(* CODESYS project PLC_Project_RECOVERED_2025-07-25T08-23-59.project

Project tree, tasks and I/O mapping:
  Device : CODESYS Control Win V3 x64, CODESYS, version 3.5.21.10
    application Application
      libraries: Standard, 3.5.18.0 (System)
      task MainTask (cyclic, interval t#20ms, priority 1) calls PLC_PRG
      section4_Method/
        function block sec4_Motor [ST]: OvldSet, StopManual, Stop, OvldReset, StartManual, Start
        program sec4_Main [ST]
      program PLC_PRG [ST]
      section2_BasicST/
        Lecture1_StandardFunction/
          program Lecture1_StandardFunction [ST]
        Exercise1/
          program Exercise1 [ST]
        Lecture2_Finite State Machine/
          program Lecture2_FiniteStateMachine [ST]
        Lecture3_Array/
          program Lecture3_Array [ST]
          function CheckFault [ST]
      section3_Class/
        Lecture1_Class/
          program POU_Class_Lecture1 [ST]
          function block Motor [ST]
          data type DUT_MotorInputVar
          data type DUT_MotorOutputVar
        Exercise1/
          data type MotorO
          data type MotorI
          program POU_Class_Exercise1 [ST]
          function block MotorEquip [ST]
*)

// Device/Application/section3_Class/Exercise1/MotorO
TYPE MotorO :
STRUCT
	Coil : BOOL;
END_STRUCT
END_TYPE

// Device/Application/section3_Class/Exercise1/MotorI
TYPE MotorI :
STRUCT
	Start : BOOL;
	Stop  : BOOL;
	OverLoad : BOOL;
	WaitTime :TIME;
 
END_STRUCT
END_TYPE

// Device/Application/section3_Class/Lecture1_Class/DUT_MotorInputVar
TYPE DUT_MotorInputVar :
	
STRUCT
	Start : BOOL;
	Stop : BOOL;
	Overload : BOOL;
END_STRUCT


END_TYPE

// Device/Application/section3_Class/Lecture1_Class/DUT_MotorOutputVar
TYPE DUT_MotorOutputVar :
	
STRUCT
	Coil : BOOL;
END_STRUCT

END_TYPE

// Device/Application/PLC_PRG
PROGRAM PLC_PRG
VAR
	Motor1 : Motor;
END_VAR

//Lecture1_StandardFunction();
//Lecture2_FiniteStateMachine();
//Lecture3_Array();
//Exercise1();
//POU_Class_Lecture1();
//POU_Class_Exercise1();
sec4_Main();

END_PROGRAM

// Device/Application/section2_BasicST/Lecture1_StandardFunction/Lecture1_StandardFunction
PROGRAM Lecture1_StandardFunction
VAR
	Start : BOOL;
	Stop : BOOL;
	Motor1 : BOOL;
	Motor2 : BOOL;
	
	Timer1 : TON;
	ElapsedTime: TIME;
	
	Reset : BOOL;
	StartTrigger : R_TRIG;
	StopTrigger : R_TRIG;
END_VAR


StartTrigger(CLK:= Start);
StopTrigger(CLK:= Stop);


IF StartTrigger.Q THEN
	Motor1 := TRUE;
END_IF


IF Motor1 THEN	
	Timer1(IN:=TRUE ,PT:=T#10S ,
	   ET=>ElapsedTime );	   
END_IF

IF Timer1.Q THEN
	Motor2 := TRUE;
END_IF
	  


IF StopTrigger.Q THEN
	Timer1(IN:=FALSE ,PT:=T#5S);	   
	Motor1 := FALSE;
	Motor2 := FALSE;
END_IF

END_PROGRAM

// Device/Application/section2_BasicST/Lecture2_Finite State Machine/Lecture2_FiniteStateMachine
PROGRAM Lecture2_FiniteStateMachine
VAR
Start : BOOL;
Stop : BOOL;

Mixer: BOOL;
Pump : BOOL;
Gate : BOOL;

Timer1 : TON;

State: INT;

StartT : R_TRIG;
StopT  : R_TRIG;

END_VAR

StartT(CLK:=Start);
StopT(CLK:=Stop);

CASE STATE OF
	0:
		Timer1(IN:=FALSE);	
		Mixer:=FALSE;
		Pump:=FALSE;
		Gate:=FALSE;
		
		IF StartT.Q THEN			
			State:=1;		
		ELSE
			State:=0;		
		END_IF
		
	1:
		Mixer:=TRUE;
		
		Timer1(IN:=TRUE , PT:=T#5S , ET=>);
		IF Timer1.Q THEN
			Timer1(IN:=FALSE);
			State:=2;
		END_IF

	2:
		Pump:=TRUE;
		
		Timer1(IN:=TRUE , PT:=T#5S , ET=>);
		IF Timer1.Q THEN
			Timer1(IN:=FALSE);	
			Pump:=FALSE;
			State:=3;		
		END_IF
		
	3:
		Timer1(IN:=TRUE , PT:=T#5S , ET=>);
		IF Timer1.Q THEN
			Timer1(IN:=FALSE);	
			Mixer:=FALSE;
			State:=4;		
		END_IF
		
	4:		
		Gate:=TRUE;
		
		Timer1(IN:=TRUE , PT:=T#3S , ET=>);
		IF Timer1.Q THEN
			Timer1(IN:=FALSE);	
			Gate:=FALSE;
			State:=0;
		END_IF
		
END_CASE


IF StopT.Q THEN
	State:=0;
END_IF

END_PROGRAM

// Device/Application/section2_BasicST/Lecture3_Array/Lecture3_Array
PROGRAM Lecture3_Array
VAR
	Buttons : ARRAY [1..4] OF BOOL;
	
	Temp : ARRAY[1..4] OF INT := [90, 20, 100, 75] ;
	OverLoad : ARRAY [1..4] OF BOOL;
	AnalogSensors : ARRAY [1..4] OF INT := [8, 2(0), 8];
	
	Coils : ARRAY [1..4] OF BOOL;
		
	i: INT;
END_VAR

FOR i:=1 TO 4 BY 1 DO
	
	IF CheckFault(Overload:=OverLoad[i] , MotorTemp:=Temp[i]) THEN
		Coils[i]:=FALSE;
	ELSIF Buttons[i]  THEN
		Coils[i]:=TRUE;
	ELSE
		Coils[i]:= FALSE;	
	END_IF
	
END_FOR

END_PROGRAM

// Device/Application/section2_BasicST/Lecture3_Array/CheckFault
FUNCTION CheckFault : BOOL
VAR_INPUT
	Overload : BOOL;
	MotorTemp : INT;
END_VAR


IF Overload OR MotorTemp>80 THEN	
	CheckFault := TRUE;
ELSE
	CheckFault := FALSE;
END_IF

END_FUNCTION

// Device/Application/section2_BasicST/Exercise1/Exercise1
PROGRAM Exercise1
VAR
	OutPumps : ARRAY [1..4] OF BOOL;
	OutPumpsFault : ARRAY [1..4] OF BOOL;
	OutValves : ARRAY [1..4] OF BOOL;
	
	InPumps : ARRAY [1..1] OF BOOL;
	InPumpsFault : ARRAY [1..1] OF BOOL;
	InValves : ARRAY [1..1] OF BOOL;
	
	LevelSensor : INT;
	
	i : INT;
	j : INT;
END_VAR



FOR i:= 1 TO 4 BY 1 DO
	OutPumps[i] := LevelSensor > 100;
END_FOR
InPumps[1] := LevelSensor <= 100;
		


//Interlog
FOR i:= 1 TO 4 BY 1 DO
	IF NOT OutValves[i] THEN
			OutPumps[i] := FALSE;		
	ELSIF CheckFault(Overload:=OutPumpsFault[i] , MotorTemp:=0) THEN
		OutPumps[i] := FALSE;	
	END_IF
	
END_FOR

IF NOT InValves[1] THEN	
	InPumps[1] := FALSE;
	
ELSIF CheckFault(Overload:=InPumpsFault[1] , MotorTemp:=0) THEN
	InPumps[1] := FALSE;
END_IF
//Interlog

END_PROGRAM

// Device/Application/section3_Class/Lecture1_Class/POU_Class_Lecture1
PROGRAM POU_Class_Lecture1
VAR
	Motors : ARRAY [1..3] OF Motor;
	MotorsI : ARRAY [1..3] OF DUT_MotorInputVar;
	MotorsO : ARRAY [1..3] OF DUT_MotorOutputVar;


	i : INT;
END_VAR


Motors[1](MotorInput:=MotorsI[1] , MotorOutput=>MotorsO[1]);
Motors[2](MotorInput:=MotorsI[2] , MotorOutput=>MotorsO[2]);
Motors[3](MotorInput:=MotorsI[3] , MotorOutput=>MotorsO[3]);

FOR i:= 1 TO 3 BY 1 DO
	MotorsI[i].Start := TRUE;
END_FOR

END_PROGRAM

// Device/Application/section3_Class/Lecture1_Class/Motor
FUNCTION_BLOCK Motor

VAR_INPUT
	MotorInput : DUT_MotorInputVar;
END_VAR

VAR_OUTPUT
	MotorOutput : DUT_MotorOutputVar;
END_VAR

VAR
	Start : BOOL;
	Stop : BOOL;
	Overload : BOOL;
	
	Coil : BOOL;
END_VAR

Start := MotorInput.Start;
Stop :=  MotorInput.Stop;
Overload := MotorInput.Overload;


IF Start AND NOT Stop AND NOT Overload THEN
	Coil := TRUE;
ELSE
	Coil := FALSE;
END_IF

MotorOutput.Coil := Coil;

END_FUNCTION_BLOCK

// Device/Application/section3_Class/Exercise1/POU_Class_Exercise1
PROGRAM POU_Class_Exercise1
VAR

Motors : ARRAY [1..NUM_MOTORS] OF MotorEquip ;
MotorInput : ARRAY[1..NUM_MOTORS] OF MotorI;
MotorOutput : ARRAY [1..NUM_MOTORS] OF MotorO;

/////////////////////Indexex////////////////////////
SerialIndex : INT:=1; ///Will be used for serial activation
Index : INT;

/////////////////////Machine Control///////Binded to HMI usually

GeneralStart : BOOL;
GeneralStop : BOOL;
ResetFault : BOOL;

///////////////////Feedback flags for the sequence status

Succed: BOOL;
Failed : BOOL;

//Detectors for STOP And Reset
StartTrig: R_TRIG;
StopTrig: R_TRIG;
ResetTrig : R_TRIG;
	 
END_VAR

VAR CONSTANT                ///////////Defien a constant as number of motors , adding a new motor is simply by increamenting this contsnt
	NUM_MOTORS : INT:=5;
END_VAR

//Assignment and Initialization
FOR  Index:=1 TO NUM_MOTORS BY 1 DO  
     MotorInput[Index].Stop:=GeneralStop; //Bind the stop button of all motors to one single generalStop  
	 MotorInput[index].WaitTime:=T#2S;  //Assign Wait time for all motors to be 3seconds
	 
	 Motors[Index](MotorInput:=MotorInput[Index] , 
					MotorOutput=>MotorOutput[Index]); //Assign IO Of every motor using a loop
END_FOR
//Assignment and Initialization


//Sequence OPeration
StartTrig(CLK:=GeneralStart); 
MotorInput[1].Start:=StartTrig.Q; //The first motor of the sequence should be assigned to the start button

IF MotorOutput[SerialIndex].Coil AND NOT Succed AND NOT Failed THEN  

		 SerialIndex := SerialIndex + 1; //If the current motor coil is activated , activate the next motor in sequence
		 
		 IF SerialIndex > NUM_MOTORS THEN
			 Succed := TRUE;
			 SerialIndex:= 1;
		 ELSE
		 	MotorInput[SerialIndex].Start := TRUE;
		 END_IF		 
	
END_IF
//Sequence OPeration

 

//Handlign Overloads
FOR Index:=1 TO NUM_MOTORS BY 1 DO //if there is ANY Overload fault then set the failed flag to TRUE
	IF MotorInput[Index].OverLoad THEN 
		Failed:=TRUE;
         EXIT;
	END_IF
END_FOR
//Handlign Overloads

//Handling Stop
StopTrig(CLK:=GeneralStop); 

IF Failed OR StopTrig.Q THEN// IF The failed flag is set to true , assign FALSE To all start signals and assign a general stop
	Succed := FALSE;
	GeneralStop := TRUE;
	SerialIndex:=1;
	
	FOR Index:=1 TO NUM_MOTORS BY 1 DO	 
			MotorInput[index].Start:=FALSE; 
	END_FOR
END_IF
//Handling Stop

//Reseting the fault
ResetTrig(CLK:=ResetFault);//If a reset fault is detected , reset the FAILED flag and Set GeneralStop to False
IF ResetTrig.Q THEN
	Failed:=FALSE;
	GeneralStop:=FALSE;
	SerialIndex:=1;
END_IF

END_PROGRAM

// Device/Application/section3_Class/Exercise1/MotorEquip
FUNCTION_BLOCK MotorEquip
VAR_INPUT
	MotorInput : MotorI;         ///Using structure as an Input
 
END_VAR

VAR_OUTPUT
		MotorOutput : MotorO;  /////Using Structure as an Output
END_VAR

VAR
	WaitTimer : TON;     ////Wait Timer
	SetReset : RS;
    RS_Output : BOOL;
END_VAR

 SetReset(SET:=MotorInput.Start , 
			RESET1:=MotorInput.Stop , 
			Q1=>RS_Output);

IF RS_Output AND NOT MotorInput.OverLoad  THEN  /////////Check if start input is activated , and there is no overload or stop button activated
	
	WaitTimer(IN:=TRUE , PT:=MotorInput.WaitTime);  ////Init the timer according to the presetTime provided and activate the timer
	IF WaitTimer.Q THEN                     /////////If preSet Time elapses turn on the motor
		MotorOutput.Coil:=TRUE;
	END_IF
	 
ELSE    ///////////If there is a stop or an overload , or start input is deactivaed , turn off the motor and deactiavte the ditmer
	WaitTimer(IN:=FALSE);
	MotorOutput.Coil:=FALSE;
END_IF

END_FUNCTION_BLOCK

// Device/Application/section4_Method/sec4_Main
PROGRAM sec4_Main
VAR
	Mode : BOOL;
	
	Motor1 : sec4_Motor;
	Motor2 : sec4_Motor;
	
	Temp : INT;
	
	OVLD1Class : BOOL;
	OVLD1 : BOOL;
	OVLD2 : BOOL;
	
	Start1 : BOOL;
	Start2 : BOOL;
	Stop1 : BOOL;
	Stop2 : BOOL;
END_VAR

Motor1(ovld:=OVLD1Class);

IF Mode THEN
	IF Temp < 100 THEN
		Motor1.Stop();
		Motor2.Stop();
	END_IF
	
	IF Temp > 100 AND Temp < 200 THEN
		Motor1.Start();
	END_IF
	
	IF Temp > 200 THEN
		Motor1.Start();
		Motor2.Start();
	END_IF
ELSE
	Motor1.StartManual(Start1);
	Motor2.StartManual(Start2);
	Motor1.StopManual(Stop1);
	Motor2.StopManual(Stop2);
END_IF


Motor1.OvldSet(ovld:= OVLD1);
Motor2.OvldSet(ovld:= OVLD2);

END_PROGRAM

// Device/Application/section4_Method/sec4_Motor
FUNCTION_BLOCK sec4_Motor
VAR_INPUT
	ovld : BOOL;
END_VAR

VAR_OUTPUT
	Coil : BOOL;
END_VAR

VAR
	FaultStatus : BOOL;
END_VAR

METHOD OvldSet : BOOL
VAR_INPUT
	ovld : BOOL;
END_VAR
IF THIS^.ovld THEN
	FaultStatus := TRUE;
	Stop();
END_IF
END_METHOD

METHOD StopManual : BOOL
VAR_INPUT
	StopB : BOOL;
END_VAR
IF StopB THEN
	Coil := FALSE;
END_IF
END_METHOD

METHOD Stop : BOOL
VAR_INPUT
END_VAR
Coil := FALSE;
END_METHOD

METHOD OvldReset : BOOL
VAR_INPUT
	ovldRst : BOOL;
END_VAR
IF ovldRst THEN
	FaultStatus := FALSE;
END_IF
END_METHOD

METHOD StartManual : BOOL
VAR_INPUT
	StartB : BOOL;
END_VAR
IF StartB THEN
	Coil := TRUE;
END_IF
END_METHOD

METHOD Start : BOOL

VAR_INPUT
	
END_VAR


Coil := TRUE;
END_METHOD

END_FUNCTION_BLOCK
